// TIA Portal V16 export
// export: Created 2024-04-05T13:37:30.8156506Z, ExportSetting WithDefaults, DisplayName Totally Integrated Automation Portal, DisplayVersion V16, DisplayName TIA Portal Version Control Interface, DisplayVersion V16, DisplayName TIA Portal Openness, DisplayVersion V16, DisplayName STEP 7 Professional, DisplayVersion V16, DisplayName STEP 7 Safety, DisplayVersion V16, DisplayName WinCC Advanced, DisplayVersion V16
VAR_GLOBAL   // PLC tag table "Default tag table"
   I_State AT %I2.0 : "UR_1_T2O_State";
   I_IO AT %I68.0 : "UR_2_T2O_IO";
   I_Joints AT %I136.0 : "UR_3_T2O_Joints";
   I_TCP AT %I240.0 : "UR_4_T2O_TCP";
   I_General_BIT AT %I34.0 : "UR_5_T2O_BitRegisters";
   I_General_INT AT %I316.0 : "UR_6_T2O_IntRegisters";
   I_General_FLOAT AT %I412.0 : "UR_6_T2O_IntRegisters";
   Q_Rotot_IO AT %Q2.0 : "UR_8_O2T_Robot_IO";
   Q_General_1 AT %Q168.0 : "UR_9_O2T_Registers";
   I_Start AT %I0.1 : Bool;
   I_Stop AT %I0.2 : Bool;
   I_Reset AT %I0.3 : Bool;
   I_Sensor2 AT %I0.4 : Bool;
   I_Sensor3 AT %I0.5 : Bool;
   I_Sensor4 AT %I0.6 : Bool;
   Q_LagerY_Omhoog AT %Q0.0 : Bool;
   Q_LagerY_Omlaag AT %Q0.1 : Bool;
   I_EStop AT %I0.7 : Bool;
   Q_Servo AT %Q1.0 : Bool;
   I_Servo AT %I1.0 : Bool;
   "VUVS-L20-P53C-MD-G18-F7-1C1" AT %I1.1 : Bool;
   Q_Geleider_Veren_Plunjer_Omhoog AT %Q0.2 : Bool;
   Q_Geleider_Veren_Plunjer_Omlaag AT %Q0.3 : Bool;
   Q_Grijper_Open AT %Q0.6 : Bool;
   Q_Grijper_Dicht AT %Q0.7 : Bool;
   Q_Plunjer_Pusher_Uit AT %Q0.4 : Bool;
   Q_Plunjer_Pusher_In AT %Q0.5 : Bool;
END_VAR
